// TIA Portal V17 program export: 1 tag tables, 0 data types, 1 data blocks, 6 code blocks (in call order from the OBs), 2 instance data blocks

VAR_GLOBAL   // PLC tag table "Default tag table"
   F_IN1 AT %I0.0 : Bool;   // SIN / CON PAR
   F_IN2 AT %I0.1 : Bool;   // LLAVIN A MAN/LOC
   F_IN3 AT %I0.2 : Bool;   // LLAVIN A AUTO/REM
   F_IN4 AT %I0.3 : Bool;   // PULSADOR OFF
   F_IN5 AT %I0.4 : Bool;   // PULSADOR MAN
   F_IN6 AT %I0.5 : Bool;   // PULSADOR AUTO
   F_IN7 AT %I0.6 : Bool;   // RES OFF
   F_IN8 AT %I0.7 : Bool;   // RES MAN
   F_IN9 AT %I1.0 : Bool;   // RES AUTO
   F_IN10 AT %I1.1 : Bool;
   F_IN11 AT %I1.2 : Bool;
   F_IN12 AT %I1.3 : Bool;
   F_IN13 AT %I1.4 : Bool;
   F_IN14 AT %I1.5 : Bool;
   F_Q1 AT %Q0.0 : Bool;   // LLAVIN ON
   F_Q2 AT %Q0.1 : Bool;   // LLAVIN AUTO
   F_Q3 AT %Q0.2 : Bool;   // PILOTO OFF
   F_Q4 AT %Q0.3 : Bool;   // PILOTO MAN
   QM1 AT %Q0.4 : Bool;   // PILOTO AUTO
   QM2 AT %Q0.5 : Bool;
   "Q0.6" AT %Q0.6 : Bool;
   "Q0.7" AT %Q0.7 : Bool;
   "Q1.0" AT %Q1.0 : Bool;
   "Q1.1" AT %Q1.1 : Bool;
   "PULSADOR OFF" AT %M0.0 : Bool;
   "PULSADOR AUTO" AT %M0.2 : Bool;
   Tag_1 AT %M200.0 : Bool;
   Tag_2 AT %M200.1 : Bool;
   Tag_3 AT %M200.3 : Bool;
   Tag_4 AT %M200.2 : Bool;
   Tag_5 AT %M200.4 : Bool;
   Tag_6 AT %M200.5 : Bool;
END_VAR

DATA_BLOCK "M"   // DB1
{ S7_Optimized_Access := 'TRUE' }
VERSION : 0.1
// stored: AutoNumber true, DBAccessibleFromOPCUA true, IsOnlyStoredInLoadMemory false, IsRetainMemResEnabled false, IsWriteProtectedInAS false, MemoryReserve 100
   VAR
      F_M1 : Bool;   // M_MODO_OFF
      F_M2 : Bool;   // M_MODO_MAN
      F_M3 : Bool;   // M_MODO_AUTO
      F_M4 : Bool;   // LLAVIN A MAN/LOC
      F_M5 : Bool;   // LLAVIN A AUTO/REM
      F_M6 : Bool;   // LLAVIN A MAN/LOC
      F_M7 : Bool;   // LLAVIN A AUTO/REM
      F_M8 : Bool;
      F_M9 : Bool;   // M_NO_RES_AUTO
      F_M10 : Bool;   // PULSADOR OFF
      F_M11 : Bool;   // PULSADOR MAN
      F_M12 : Bool;   // PULSADOR AUTO
      F_M13 : Bool;   // NO PULSADOR OFF
      F_M14 : Bool;   // NO PULSADOR MAN
      F_M15 : Bool;   // NO PULSADOR AUTO
      F_M16 : Bool;   // RES OFF
      F_M17 : Bool;   // RES MAN
      F_M18 : Bool;   // RES AUTO
      F_M19 : Bool;   // NO RES OFF
      F_M20 : Bool;   // NO RES MAN
   END_VAR
BEGIN
END_DATA_BLOCK

ORGANIZATION_BLOCK "Main"   // OB1, LAD, ProgramCycle
TITLE = "Main Program Sweep (Cycle)"
{ S7_Optimized_Access := 'TRUE' }
VERSION : 0.1
// stored: AutoNumber true, IsIECCheckEnabled false, SetENOAutomatically false
   VAR_INPUT
      Initial_Call : Bool;   // Initial call of this OB
      Remanence : Bool;   // =True, if remanent data are available
   END_VAR
BEGIN
END_ORGANIZATION_BLOCK

FUNCTION "Llavin Filtrado" : Void   // FC3, LAD
{ S7_Optimized_Access := 'TRUE' }
VERSION : 0.1
// stored: AutoNumber true, IsIECCheckEnabled false, SetENOAutomatically false, UDAEnableTagReadback false
BEGIN

REGION Network 1: LLAVIN A MAN/LOC
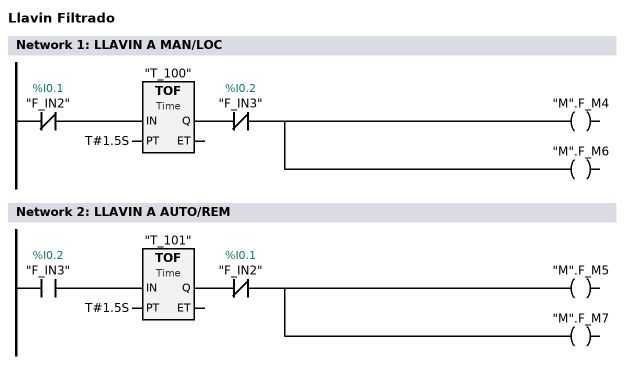
   RUNG wire#powerrail
      I_Contact( "F_IN2" )
      { S7_Templates := "time_type := Time" } "T_100".TOF(pt := T#1.5S, et =>)
      I_Contact( "F_IN3" )
      wire#w1
      Coil( "M".F_M4 )
   END_RUNG
   RUNG wire#w1
      Coil( "M".F_M6 )
   END_RUNG
   // the same network as SCL:
   "T_100".TOF(IN := NOT "F_IN2", PT := T#1.5S);
   "M".F_M4 := "T_100".Q AND NOT "F_IN3";
   "M".F_M6 := "M".F_M4;
END_REGION

REGION Network 2: LLAVIN A AUTO/REM
   RUNG wire#powerrail
      Contact( "F_IN3" )
      { S7_Templates := "time_type := Time" } "T_101".TOF(pt := T#1.5S, et =>)
      I_Contact( "F_IN2" )
      wire#w1
      Coil( "M".F_M5 )
   END_RUNG
   RUNG wire#w1
      Coil( "M".F_M7 )
   END_RUNG
   // the same network as SCL:
   "T_101".TOF(IN := "F_IN3", PT := T#1.5S);
   "M".F_M5 := "T_101".Q AND NOT "F_IN2";
   "M".F_M7 := "M".F_M5;
END_REGION
END_FUNCTION

FUNCTION "Logica" : Void   // FC4, LAD
{ S7_Optimized_Access := 'TRUE' }
VERSION : 0.1
// stored: AutoNumber true, IsIECCheckEnabled false, SetENOAutomatically false, UDAEnableTagReadback false
BEGIN

REGION Network 1: M_MODO_OFF
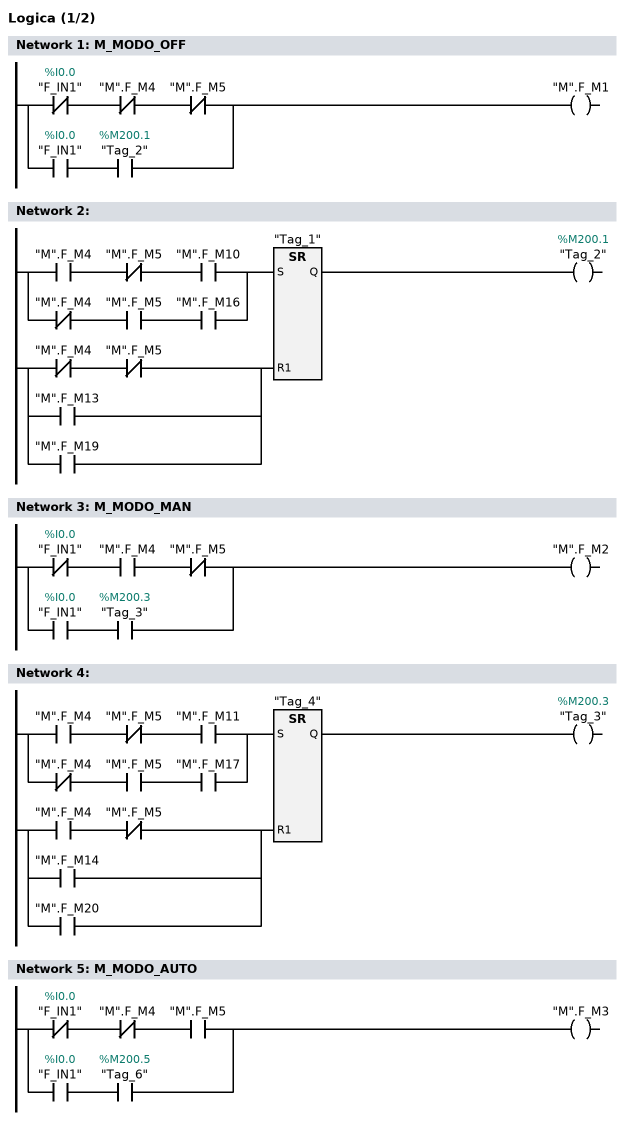
   RUNG wire#powerrail
      I_Contact( "F_IN1" )
      I_Contact( "M".F_M4 )
      I_Contact( "M".F_M5 )
      wire#w1
      Coil( "M".F_M1 )
   END_RUNG
   RUNG wire#powerrail
      Contact( "F_IN1" )
      Contact( "Tag_2" )
   END_RUNG wire#w1
   // the same network as SCL:
   "M".F_M1 := (NOT "F_IN1" AND NOT "M".F_M4 AND NOT "M".F_M5) OR ("F_IN1" AND "Tag_2");
END_REGION

REGION Network 2
   RUNG wire#powerrail
      Contact( "M".F_M4 )
      I_Contact( "M".F_M5 )
      Contact( "M".F_M10 )
      wire#w1
      S_SR(operand := "Tag_1", r1 := wire#w2)
      Coil( "Tag_2" )
   END_RUNG
   RUNG wire#powerrail
      I_Contact( "M".F_M4 )
      Contact( "M".F_M5 )
      Contact( "M".F_M16 )
   END_RUNG wire#w1
   RUNG wire#powerrail
      I_Contact( "M".F_M4 )
      I_Contact( "M".F_M5 )
   END_RUNG wire#w2
   RUNG wire#powerrail
      Contact( "M".F_M13 )
   END_RUNG wire#w2
   RUNG wire#powerrail
      Contact( "M".F_M19 )
   END_RUNG wire#w2
   // the same network as SCL:
   IF ("M".F_M4 AND NOT "M".F_M5 AND "M".F_M10) OR (NOT "M".F_M4 AND "M".F_M5 AND "M".F_M16) THEN
       "Tag_1" := TRUE;   // SR flip-flop
   END_IF;
   IF (NOT "M".F_M4 AND NOT "M".F_M5) OR "M".F_M13 OR "M".F_M19 THEN "Tag_1" := FALSE; END_IF;
   "Tag_2" := "Tag_1";
END_REGION

REGION Network 3: M_MODO_MAN
   RUNG wire#powerrail
      I_Contact( "F_IN1" )
      Contact( "M".F_M4 )
      I_Contact( "M".F_M5 )
      wire#w1
      Coil( "M".F_M2 )
   END_RUNG
   RUNG wire#powerrail
      Contact( "F_IN1" )
      Contact( "Tag_3" )
   END_RUNG wire#w1
   // the same network as SCL:
   "M".F_M2 := (NOT "F_IN1" AND "M".F_M4 AND NOT "M".F_M5) OR ("F_IN1" AND "Tag_3");
END_REGION

REGION Network 4
   RUNG wire#powerrail
      Contact( "M".F_M4 )
      I_Contact( "M".F_M5 )
      Contact( "M".F_M11 )
      wire#w1
      S_SR(operand := "Tag_4", r1 := wire#w2)
      Coil( "Tag_3" )
   END_RUNG
   RUNG wire#powerrail
      I_Contact( "M".F_M4 )
      Contact( "M".F_M5 )
      Contact( "M".F_M17 )
   END_RUNG wire#w1
   RUNG wire#powerrail
      Contact( "M".F_M4 )
      I_Contact( "M".F_M5 )
   END_RUNG wire#w2
   RUNG wire#powerrail
      Contact( "M".F_M14 )
   END_RUNG wire#w2
   RUNG wire#powerrail
      Contact( "M".F_M20 )
   END_RUNG wire#w2
   // the same network as SCL:
   IF ("M".F_M4 AND NOT "M".F_M5 AND "M".F_M11) OR (NOT "M".F_M4 AND "M".F_M5 AND "M".F_M17) THEN
       "Tag_4" := TRUE;   // SR flip-flop
   END_IF;
   IF ("M".F_M4 AND NOT "M".F_M5) OR "M".F_M14 OR "M".F_M20 THEN "Tag_4" := FALSE; END_IF;
   "Tag_3" := "Tag_4";
END_REGION

REGION Network 5: M_MODO_AUTO
   RUNG wire#powerrail
      I_Contact( "F_IN1" )
      I_Contact( "M".F_M4 )
      Contact( "M".F_M5 )
      wire#w1
      Coil( "M".F_M3 )
   END_RUNG
   RUNG wire#powerrail
      Contact( "F_IN1" )
      Contact( "Tag_6" )
   END_RUNG wire#w1
   // the same network as SCL:
   "M".F_M3 := (NOT "F_IN1" AND NOT "M".F_M4 AND "M".F_M5) OR ("F_IN1" AND "Tag_6");
END_REGION

REGION Network 6
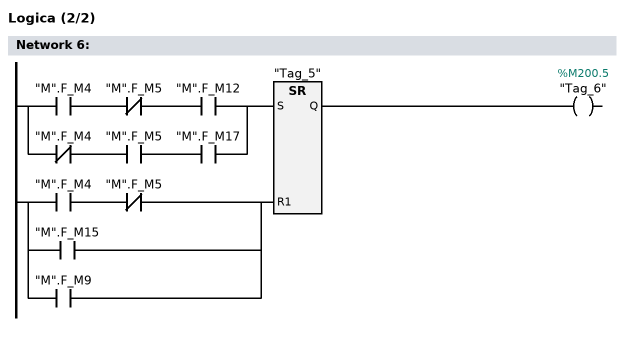
   RUNG wire#powerrail
      Contact( "M".F_M4 )
      I_Contact( "M".F_M5 )
      Contact( "M".F_M12 )
      wire#w1
      S_SR(operand := "Tag_5", r1 := wire#w2)
      Coil( "Tag_6" )
   END_RUNG
   RUNG wire#powerrail
      I_Contact( "M".F_M4 )
      Contact( "M".F_M5 )
      Contact( "M".F_M17 )
   END_RUNG wire#w1
   RUNG wire#powerrail
      Contact( "M".F_M4 )
      I_Contact( "M".F_M5 )
   END_RUNG wire#w2
   RUNG wire#powerrail
      Contact( "M".F_M15 )
   END_RUNG wire#w2
   RUNG wire#powerrail
      Contact( "M".F_M9 )
   END_RUNG wire#w2
   // the same network as SCL:
   IF ("M".F_M4 AND NOT "M".F_M5 AND "M".F_M12) OR (NOT "M".F_M4 AND "M".F_M5 AND "M".F_M17) THEN
       "Tag_5" := TRUE;   // SR flip-flop
   END_IF;
   IF ("M".F_M4 AND NOT "M".F_M5) OR "M".F_M15 OR "M".F_M9 THEN "Tag_5" := FALSE; END_IF;
   "Tag_6" := "Tag_5";
END_REGION
END_FUNCTION

FUNCTION "Pulsadores" : Void   // FC2, LAD
{ S7_Optimized_Access := 'TRUE' }
VERSION : 0.1
// stored: AutoNumber true, IsIECCheckEnabled false, SetENOAutomatically false, UDAEnableTagReadback false
BEGIN

REGION Network 1: PULSADOR OFF
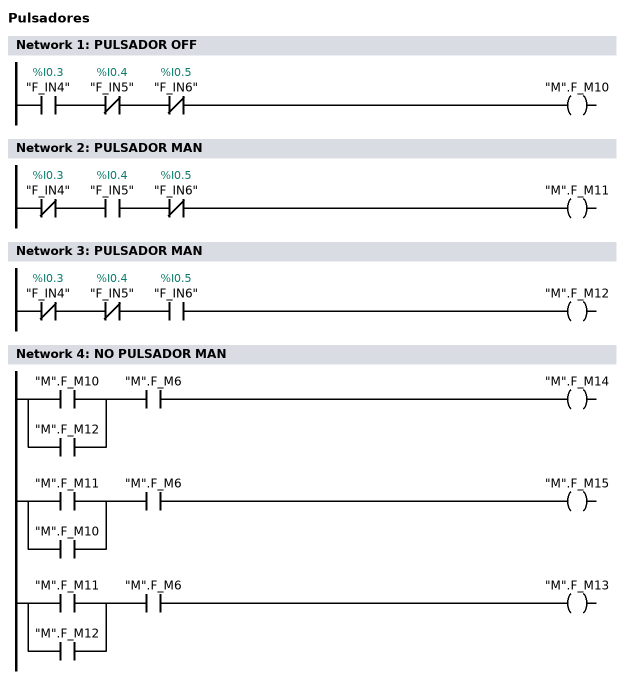
   RUNG wire#powerrail
      Contact( "F_IN4" )
      I_Contact( "F_IN5" )
      I_Contact( "F_IN6" )
      Coil( "M".F_M10 )
   END_RUNG
   // the same network as SCL:
   "M".F_M10 := "F_IN4" AND NOT "F_IN5" AND NOT "F_IN6";
END_REGION

REGION Network 2: PULSADOR MAN
   RUNG wire#powerrail
      I_Contact( "F_IN4" )
      Contact( "F_IN5" )
      I_Contact( "F_IN6" )
      Coil( "M".F_M11 )
   END_RUNG
   // the same network as SCL:
   "M".F_M11 := NOT "F_IN4" AND "F_IN5" AND NOT "F_IN6";
END_REGION

REGION Network 3: PULSADOR MAN
   RUNG wire#powerrail
      I_Contact( "F_IN4" )
      I_Contact( "F_IN5" )
      Contact( "F_IN6" )
      Coil( "M".F_M12 )
   END_RUNG
   // the same network as SCL:
   "M".F_M12 := NOT "F_IN4" AND NOT "F_IN5" AND "F_IN6";
END_REGION

REGION Network 4: NO PULSADOR MAN
   RUNG wire#powerrail
      Contact( "M".F_M10 )
      wire#w1
      Contact( "M".F_M6 )
      Coil( "M".F_M14 )
   END_RUNG
   RUNG wire#powerrail
      Contact( "M".F_M12 )
   END_RUNG wire#w1
   RUNG wire#powerrail
      Contact( "M".F_M11 )
      wire#w2
      Contact( "M".F_M6 )
      Coil( "M".F_M15 )
   END_RUNG
   RUNG wire#powerrail
      Contact( "M".F_M10 )
   END_RUNG wire#w2
   RUNG wire#powerrail
      Contact( "M".F_M11 )
      wire#w3
      Contact( "M".F_M6 )
      Coil( "M".F_M13 )
   END_RUNG
   RUNG wire#powerrail
      Contact( "M".F_M12 )
   END_RUNG wire#w3
   // the same network as SCL:
   "M".F_M14 := ("M".F_M10 OR "M".F_M12) AND "M".F_M6;
   "M".F_M15 := ("M".F_M11 OR "M".F_M10) AND "M".F_M6;
   "M".F_M13 := ("M".F_M11 OR "M".F_M12) AND "M".F_M6;
END_REGION
END_FUNCTION

FUNCTION "Res" : Void   // FC1, LAD
{ S7_Optimized_Access := 'TRUE' }
VERSION : 0.1
// stored: AutoNumber true, IsIECCheckEnabled false, SetENOAutomatically false, UDAEnableTagReadback false
BEGIN

REGION Network 1: PULSADOR OFF
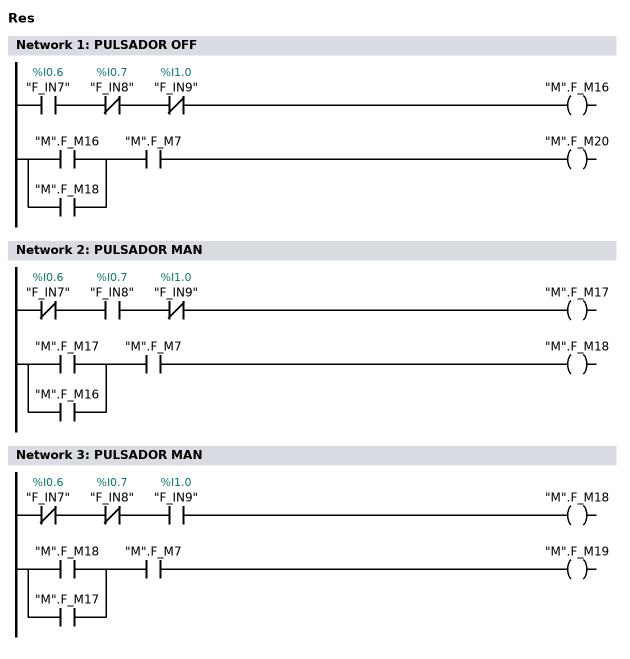
   RUNG wire#powerrail
      Contact( "F_IN7" )
      I_Contact( "F_IN8" )
      I_Contact( "F_IN9" )
      Coil( "M".F_M16 )
   END_RUNG
   RUNG wire#powerrail
      Contact( "M".F_M16 )
      wire#w1
      Contact( "M".F_M7 )
      Coil( "M".F_M20 )
   END_RUNG
   RUNG wire#powerrail
      Contact( "M".F_M18 )
   END_RUNG wire#w1
   // the same network as SCL:
   "M".F_M16 := "F_IN7" AND NOT "F_IN8" AND NOT "F_IN9";
   "M".F_M20 := ("M".F_M16 OR "M".F_M18) AND "M".F_M7;
END_REGION

REGION Network 2: PULSADOR MAN
   RUNG wire#powerrail
      I_Contact( "F_IN7" )
      Contact( "F_IN8" )
      I_Contact( "F_IN9" )
      Coil( "M".F_M17 )
   END_RUNG
   RUNG wire#powerrail
      Contact( "M".F_M17 )
      wire#w1
      Contact( "M".F_M7 )
      Coil( "M".F_M18 )
   END_RUNG
   RUNG wire#powerrail
      Contact( "M".F_M16 )
   END_RUNG wire#w1
   // the same network as SCL:
   "M".F_M17 := NOT "F_IN7" AND "F_IN8" AND NOT "F_IN9";
   "M".F_M18 := ("M".F_M17 OR "M".F_M16) AND "M".F_M7;
END_REGION

REGION Network 3: PULSADOR MAN
   RUNG wire#powerrail
      I_Contact( "F_IN7" )
      I_Contact( "F_IN8" )
      Contact( "F_IN9" )
      Coil( "M".F_M18 )
   END_RUNG
   RUNG wire#powerrail
      Contact( "M".F_M18 )
      wire#w1
      Contact( "M".F_M7 )
      Coil( "M".F_M19 )
   END_RUNG
   RUNG wire#powerrail
      Contact( "M".F_M17 )
   END_RUNG wire#w1
   // the same network as SCL:
   "M".F_M18 := NOT "F_IN7" AND NOT "F_IN8" AND "F_IN9";
   "M".F_M19 := ("M".F_M18 OR "M".F_M17) AND "M".F_M7;
END_REGION
END_FUNCTION

FUNCTION "Salidas" : Void   // FC5, LAD
{ S7_Optimized_Access := 'TRUE' }
VERSION : 0.1
// stored: AutoNumber true, IsIECCheckEnabled false, SetENOAutomatically false, UDAEnableTagReadback false
BEGIN

REGION Network 1: PILOTO OFF
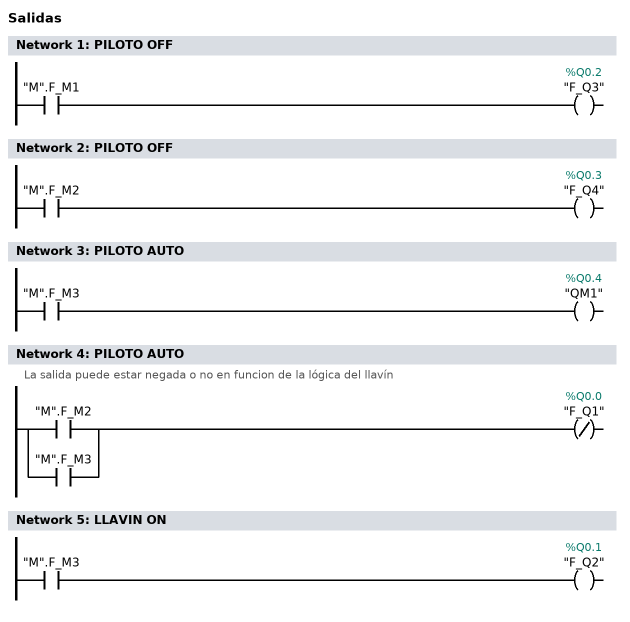
   RUNG wire#powerrail
      Contact( "M".F_M1 )
      Coil( "F_Q3" )
   END_RUNG
   // the same network as SCL:
   "F_Q3" := "M".F_M1;
END_REGION

REGION Network 2: PILOTO OFF
   RUNG wire#powerrail
      Contact( "M".F_M2 )
      Coil( "F_Q4" )
   END_RUNG
   // the same network as SCL:
   "F_Q4" := "M".F_M2;
END_REGION

REGION Network 3: PILOTO AUTO
   RUNG wire#powerrail
      Contact( "M".F_M3 )
      Coil( "QM1" )
   END_RUNG
   // the same network as SCL:
   "QM1" := "M".F_M3;
END_REGION

REGION Network 4: PILOTO AUTO
   // La salida puede estar negada o no en funcion de la lógica del llavín
   RUNG wire#powerrail
      Contact( "M".F_M2 )
      wire#w1
      I_Coil( "F_Q1" )
   END_RUNG
   RUNG wire#powerrail
      Contact( "M".F_M3 )
   END_RUNG wire#w1
   // the same network as SCL:
   "F_Q1" := NOT ("M".F_M2 OR "M".F_M3);
END_REGION

REGION Network 5: LLAVIN ON
   RUNG wire#powerrail
      Contact( "M".F_M3 )
      Coil( "F_Q2" )
   END_RUNG
   // the same network as SCL:
   "F_Q2" := "M".F_M3;
END_REGION
END_FUNCTION

DATA_BLOCK "T_100"   // DB100
{ S7_Optimized_Access := 'TRUE' }
// stored: AutoNumber false, DBAccessibleFromOPCUA true, InstanceOfName IEC_TIMER, OfSystemLibElement IEC_TIMER, OfSystemLibVersion 1.0
"IEC_TIMER"
   // VAR
   //    PT : Time;
   //    ET { ExternalWritable := 'False'} : Time;
   //    IN : Bool;
   //    Q { ExternalWritable := 'False'} : Bool;
   // END_VAR
BEGIN
END_DATA_BLOCK

DATA_BLOCK "T_101"   // DB101
{ S7_Optimized_Access := 'TRUE' }
// stored: AutoNumber false, DBAccessibleFromOPCUA true, InstanceOfName IEC_TIMER, OfSystemLibElement IEC_TIMER, OfSystemLibVersion 1.0
"IEC_TIMER"
   // VAR
   //    PT : Time;
   //    ET { ExternalWritable := 'False'} : Time;
   //    IN : Bool;
   //    Q { ExternalWritable := 'False'} : Bool;
   // END_VAR
BEGIN
END_DATA_BLOCK
